% RSLogix 500 project DDE-Messaging.RSS, saved by version 8.40.00.08 %
PROJECT "UNTITLED"    % processor: Bul.1763 MicroLogix 1100 Series B %

PROGRAM FILES
  LAD 2   4 rungs
  LAD 3 "CTRL"  10 rungs
  LAD 4 "STRINGS"  6 rungs
  LAD 5 "COUNTERS"  9 rungs

DATA FILES
  O0 OUTPUT  4 elements
  I1 INPUT  6 elements
  S2 STATUS  66 elements
  B3 BINARY  1 elements
  T4 TIMER  4 elements
  C5 COUNTER  4 elements
  R6 CONTROL  1 elements
  N7 INTEGER  4 elements
  F8 FLOAT  1 elements
  ST9   7 elements

LADDER 2
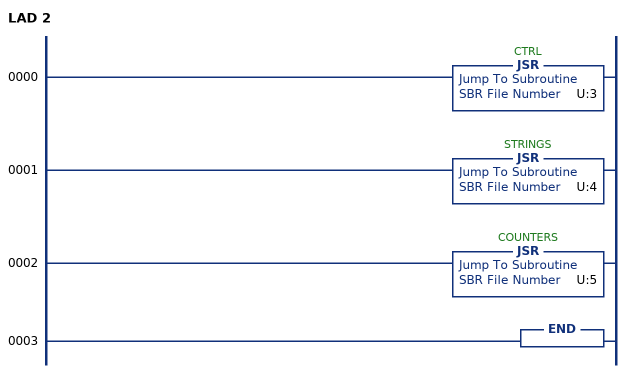
% Rung: 0 %
SOR JSR U:3 EOR
%   U:3  "CTRL" %
% Rung: 1 %
SOR JSR U:4 EOR
%   U:4  "STRINGS" %
% Rung: 2 %
SOR JSR U:5 EOR
%   U:5  "COUNTERS" %
% Rung: 3 %
SOR END EOR

LADDER 3 "CTRL"
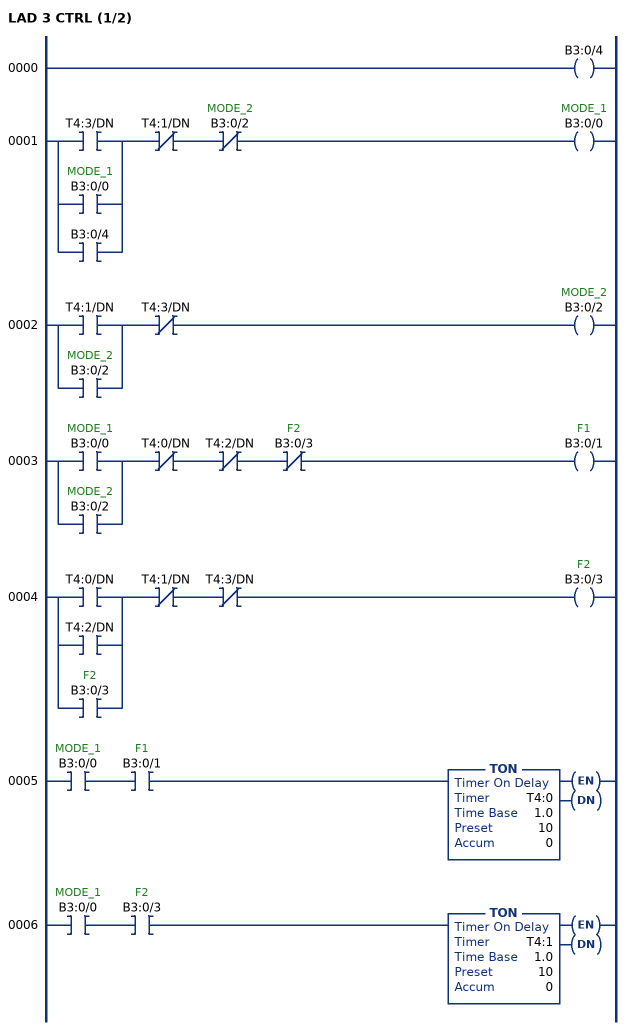
% Rung: 0 %
SOR OTE B3:0/4 EOR
% Rung: 1 %
SOR BST XIC T4:3/DN NXB XIC B3:0/0 NXB XIC B3:0/4 BND XIO T4:1/DN XIO B3:0/2 OTE B3:0/0 EOR
%   B3:0/0  MODE_1 %
%   B3:0/2  MODE_2 %
% Rung: 2 %
SOR BST XIC T4:1/DN NXB XIC B3:0/2 BND XIO T4:3/DN OTE B3:0/2 EOR
%   B3:0/2  MODE_2 %
% Rung: 3 %
SOR BST XIC B3:0/0 NXB XIC B3:0/2 BND XIO T4:0/DN XIO T4:2/DN XIO B3:0/3 OTE B3:0/1 EOR
%   B3:0/0  MODE_1 %
%   B3:0/2  MODE_2 %
%   B3:0/3  F2 %
%   B3:0/1  F1 %
% Rung: 4 %
SOR BST XIC T4:0/DN NXB XIC T4:2/DN NXB XIC B3:0/3 BND XIO T4:1/DN XIO T4:3/DN OTE B3:0/3 EOR
%   B3:0/3  F2 %
% Rung: 5 %
SOR XIC B3:0/0 XIC B3:0/1 TON T4:0 1.0 10 0 EOR
%   B3:0/0  MODE_1 %
%   B3:0/1  F1 %
% Rung: 6 %
SOR XIC B3:0/0 XIC B3:0/3 TON T4:1 1.0 10 0 EOR
%   B3:0/0  MODE_1 %
%   B3:0/3  F2 %

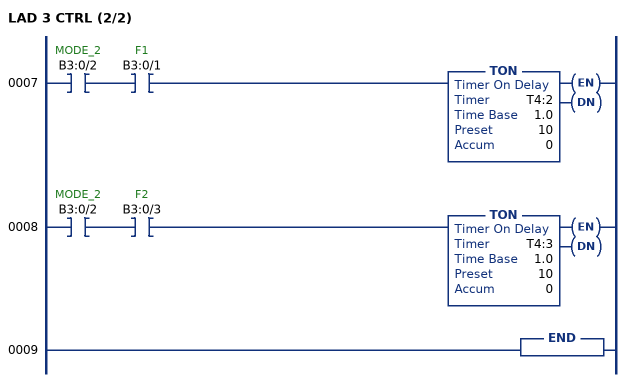
% Rung: 7 %
SOR XIC B3:0/2 XIC B3:0/1 TON T4:2 1.0 10 0 EOR
%   B3:0/2  MODE_2 %
%   B3:0/1  F1 %
% Rung: 8 %
SOR XIC B3:0/2 XIC B3:0/3 TON T4:3 1.0 10 0 EOR
%   B3:0/2  MODE_2 %
%   B3:0/3  F2 %
% Rung: 9 %
SOR END EOR

LADDER 4 "STRINGS"
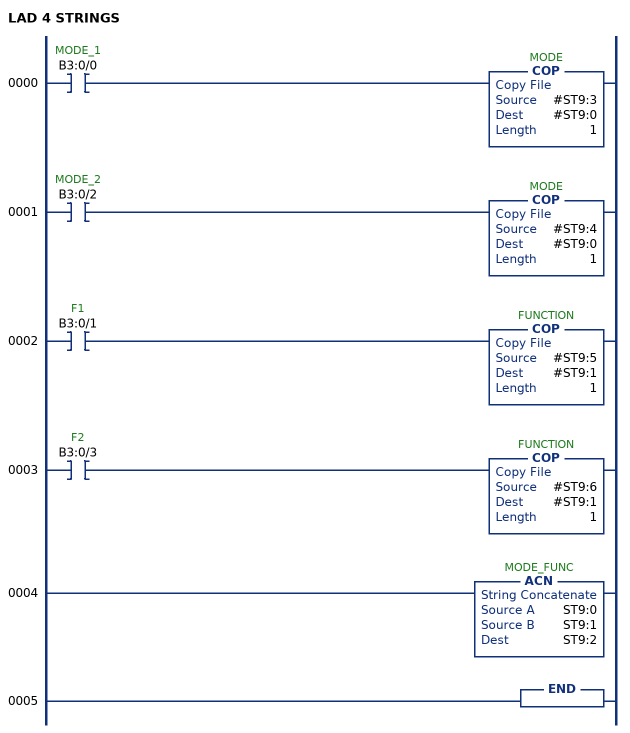
% Rung: 0 %
SOR XIC B3:0/0 COP #ST9:3 #ST9:0 1 EOR
%   B3:0/0  MODE_1 %
%   ST9:0  MODE %
% Rung: 1 %
SOR XIC B3:0/2 COP #ST9:4 #ST9:0 1 EOR
%   B3:0/2  MODE_2 %
%   ST9:0  MODE %
% Rung: 2 %
SOR XIC B3:0/1 COP #ST9:5 #ST9:1 1 EOR
%   B3:0/1  F1 %
%   ST9:1  FUNCTION %
% Rung: 3 %
SOR XIC B3:0/3 COP #ST9:6 #ST9:1 1 EOR
%   B3:0/3  F2 %
%   ST9:1  FUNCTION %
% Rung: 4 %
SOR ACN ST9:0 ST9:1 ST9:2 EOR
%   ST9:0  MODE %
%   ST9:1  FUNCTION %
%   ST9:2  MODE_FUNC %
% Rung: 5 %
SOR END EOR

LADDER 5 "COUNTERS"
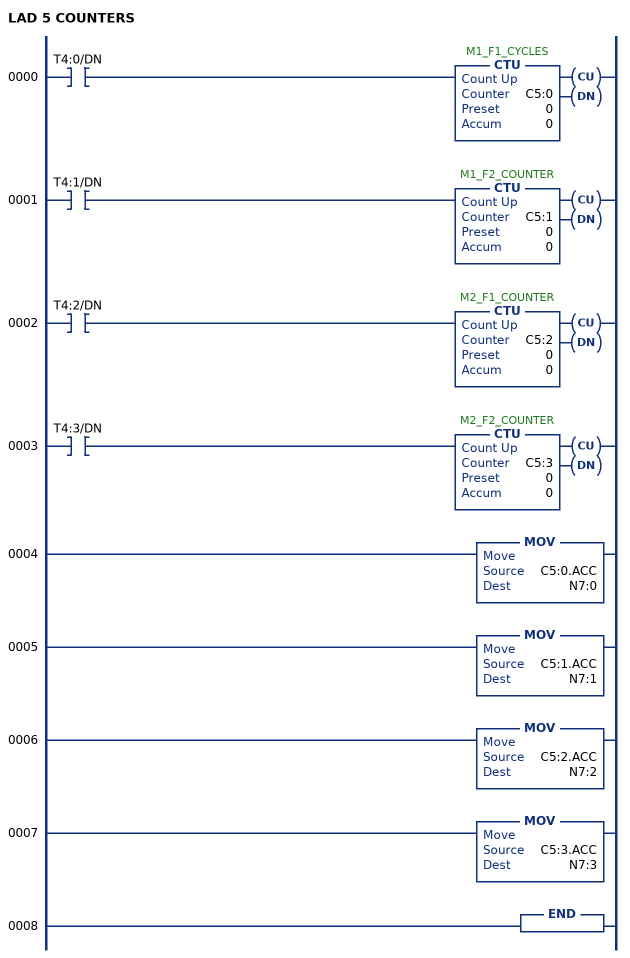
% Rung: 0 %
SOR XIC T4:0/DN CTU C5:0 0 0 EOR
%   C5:0  M1_F1_CYCLES %
% Rung: 1 %
SOR XIC T4:1/DN CTU C5:1 0 0 EOR
%   C5:1  M1_F2_COUNTER %
% Rung: 2 %
SOR XIC T4:2/DN CTU C5:2 0 0 EOR
%   C5:2  M2_F1_COUNTER %
% Rung: 3 %
SOR XIC T4:3/DN CTU C5:3 0 0 EOR
%   C5:3  M2_F2_COUNTER %
% Rung: 4 %
SOR MOV C5:0.ACC N7:0 EOR
%   C5:0  M1_F1_CYCLES %
% Rung: 5 %
SOR MOV C5:1.ACC N7:1 EOR
%   C5:1  M1_F2_COUNTER %
% Rung: 6 %
SOR MOV C5:2.ACC N7:2 EOR
%   C5:2  M2_F1_COUNTER %
% Rung: 7 %
SOR MOV C5:3.ACC N7:3 EOR
%   C5:3  M2_F2_COUNTER %
% Rung: 8 %
SOR END EOR

DATA TABLE (non-zero values as saved)
DATA T4
% .PRE .ACC %
% T4:0 % 10 0
% T4:1 % 10 0
% T4:2 % 10 0
% T4:3 % 10 0
DATA ST9
% ST9:3 % "MODE-1"
% ST9:4 % "MODE-2"
% ST9:5 % "F-1"
% ST9:6 % "F-2"
